// TIA Portal V18 export
FUNCTION "ST10_Device" : Void   // FC1010, LAD
{ S7_Optimized_Access := 'TRUE' }
// stored: AutoNumber false, SetENOAutomatically false
   VAR_INPUT
      iSysMode : "RCS_SysComInterface_V1";
   END_VAR
BEGIN

NETWORK
TITLE = SafetyGate

      CALL  "ST10_SafetyGate"
      ( iSysMode := #iSysMode
      );


NETWORK
TITLE = PartData

      CALL  "ST10_PartData"
      ( iSysMode := #iSysMode
      );


NETWORK
TITLE = Analog

      CALL  "ST10_Analog"
      ( iSysMode := #iSysMode
      );


REGION Network 4: SR Scan
END_REGION

REGION Network 7: CuringOven
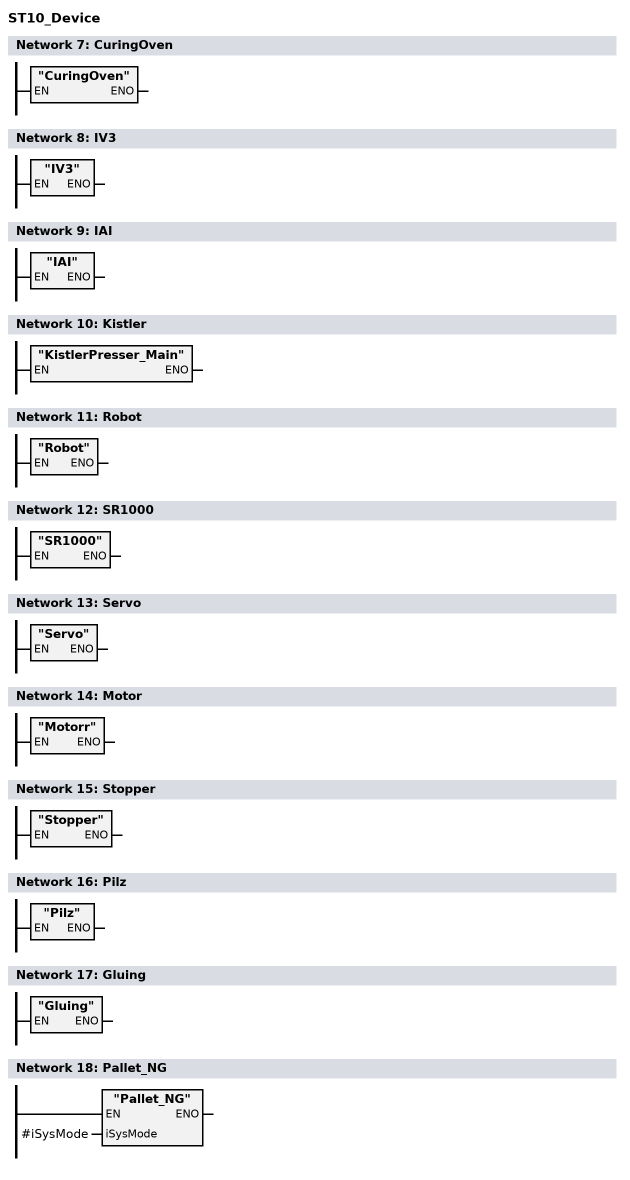
   RUNG wire#powerrail
      "CuringOven"()
   END_RUNG
   // the same network as SCL:
   "CuringOven"();
END_REGION

REGION Network 8: IV3
   RUNG wire#powerrail
      "IV3"()
   END_RUNG
   // the same network as SCL:
   "IV3"();
END_REGION

REGION Network 9: IAI
   RUNG wire#powerrail
      "IAI"()
   END_RUNG
   // the same network as SCL:
   "IAI"();
END_REGION

REGION Network 10: Kistler
   RUNG wire#powerrail
      "KistlerPresser_Main"()
   END_RUNG
   // the same network as SCL:
   "KistlerPresser_Main"();
END_REGION

REGION Network 11: Robot
   RUNG wire#powerrail
      "Robot"()
   END_RUNG
   // the same network as SCL:
   "Robot"();
END_REGION

REGION Network 12: SR1000
   RUNG wire#powerrail
      "SR1000"()
   END_RUNG
   // the same network as SCL:
   "SR1000"();
END_REGION

REGION Network 13: Servo
   RUNG wire#powerrail
      "Servo"()
   END_RUNG
   // the same network as SCL:
   "Servo"();
END_REGION

REGION Network 14: Motor
   RUNG wire#powerrail
      "Motorr"()
   END_RUNG
   // the same network as SCL:
   "Motorr"();
END_REGION

REGION Network 15: Stopper
   RUNG wire#powerrail
      "Stopper"()
   END_RUNG
   // the same network as SCL:
   "Stopper"();
END_REGION

REGION Network 16: Pilz
   RUNG wire#powerrail
      "Pilz"()
   END_RUNG
   // the same network as SCL:
   "Pilz"();
END_REGION

REGION Network 17: Gluing
   RUNG wire#powerrail
      "Gluing"()
   END_RUNG
   // the same network as SCL:
   "Gluing"();
END_REGION

REGION Network 18: Pallet_NG
   RUNG wire#powerrail
      "Pallet_NG"(iSysMode := #iSysMode)
   END_RUNG
   // the same network as SCL:
   "Pallet_NG"(iSysMode := #iSysMode);
END_REGION
END_FUNCTION
